// TIA Portal V20 export
FUNCTION_BLOCK "FB_Axis"   // FB30140, LAD
{ S7_Optimized_Access := 'TRUE' }
// stored: AutoNumber false, MemoryReserve 100, SetENOAutomatically false
   VAR_INPUT
      TO_PosAxis : TO_PositioningAxis;
      I_bMan_Enable : Bool;
      I_iHomeMode : Int;
      I_iHomePos : LReal;
   END_VAR
   VAR_IN_OUT
      Ds_Axis : "sAxis";
   END_VAR
   VAR
      instAxis01 { ExternalAccessible := 'False'; ExternalVisible := 'False'; ExternalWritable := 'False'} : "LAxisCtrl_PosAxis";
      instShearAxisStatus { S7_SetPoint := 'True'} : "LAxisCtrl_GetAxisStatusWord";
      RT_Reset { S7_SetPoint := 'True'} : R_TRIG;
      RT_PB { ExternalAccessible := 'False'; ExternalVisible := 'False'; ExternalWritable := 'False'} : Array[0..19] of R_TRIG;   // Störungen / Alarms
      FT_PB { ExternalAccessible := 'False'; ExternalVisible := 'False'; ExternalWritable := 'False'; S7_SetPoint := 'True'} : Array[0..19] of F_TRIG;   // Störungen unterdrücken, Belegung identisch mit "Alarm" / Hide Alarms, identical with "Alarm"
      TON_PB { ExternalAccessible := 'False'; ExternalVisible := 'False'; ExternalWritable := 'False'} : Array[0..19] of TON_TIME;   // Fallende Flanke / Falling edge
      TOF_PB { ExternalAccessible := 'False'; ExternalVisible := 'False'; ExternalWritable := 'False'} : Array[0..19] of TOF_TIME;   // Negativer Impuls / Negative pulse
      i { S7_SetPoint := 'True'} : Int;
      temp_cmd_bEnableAxis { ExternalAccessible := 'False'; ExternalVisible := 'False'; ExternalWritable := 'False'} : Bool;
      temp_cmd_bresetAxis { ExternalAccessible := 'False'; ExternalVisible := 'False'; ExternalWritable := 'False'} : Bool;
      temp_cmd_bjogForward { ExternalAccessible := 'False'; ExternalVisible := 'False'; ExternalWritable := 'False'} : Bool;
      temp_cmd_bjogBackward { ExternalAccessible := 'False'; ExternalVisible := 'False'; ExternalWritable := 'False'} : Bool;
      temp_cmd_bmoveVelocity { ExternalAccessible := 'False'; ExternalVisible := 'False'; ExternalWritable := 'False'} : Bool;
      temp_cmd_bstop { ExternalAccessible := 'False'; ExternalVisible := 'False'; ExternalWritable := 'False'} : Bool;
      temp_cmd_bfastStop { ExternalAccessible := 'False'; ExternalVisible := 'False'; ExternalWritable := 'False'} : Bool;
      temp_cmd_bhoming { ExternalAccessible := 'False'; ExternalVisible := 'False'; ExternalWritable := 'False'} : Bool;
      temp_cmd_bGoToPos { ExternalAccessible := 'False'; ExternalVisible := 'False'; ExternalWritable := 'False'} : Array[0..16] of Bool;
      temp_cmd_iGoToPos : Word;
      temp_cmd_bCallAbsPos : Bool;
      temp_cmd_bRelPos : Bool;
      temp_Para_rJog_Speed { ExternalAccessible := 'False'; ExternalVisible := 'False'; ExternalWritable := 'False'} : LReal;
      temp_cmd_bGoToPosAll { ExternalAccessible := 'False'; ExternalVisible := 'False'; ExternalWritable := 'False'} : Bool;
      temp_configuration { ExternalAccessible := 'False'; ExternalVisible := 'False'; ExternalWritable := 'False'} : "LAxisCtrl_typeAxisConfig";   // Diagnostics structure
      temp_Status { ExternalAccessible := 'False'; ExternalVisible := 'False'; ExternalWritable := 'False'} : Word;
      tempAxisEnabled { ExternalAccessible := 'False'; ExternalVisible := 'False'; ExternalWritable := 'False'} : Bool;
      temp_CommandBusy { ExternalAccessible := 'False'; ExternalVisible := 'False'; ExternalWritable := 'False'} : Bool;
      temp_CommandDone { ExternalAccessible := 'False'; ExternalVisible := 'False'; ExternalWritable := 'False'} : Bool;
      temp_CommandAborted { ExternalAccessible := 'False'; ExternalVisible := 'False'; ExternalWritable := 'False'} : Bool;
      temp_InVelocity { ExternalAccessible := 'False'; ExternalVisible := 'False'; ExternalWritable := 'False'} : Bool;
      temp_jogSelected { ExternalAccessible := 'False'; ExternalVisible := 'False'; ExternalWritable := 'False'} : Bool;
      tempPosAbsoluteSelected { ExternalAccessible := 'False'; ExternalVisible := 'False'; ExternalWritable := 'False'} : Bool;
      temp_diagnostics { ExternalAccessible := 'False'; ExternalVisible := 'False'; ExternalWritable := 'False'} : "LAxisCtrl_typeDiagnostics";
      temp_stop_Dec { ExternalAccessible := 'False'; ExternalVisible := 'False'; ExternalWritable := 'False'} : LReal;
      temp_faststop_Dec { ExternalAccessible := 'False'; ExternalVisible := 'False'; ExternalWritable := 'False'} : LReal;
      temp_iFBStatus : Word;
      temp_iMCStatus : Word;
      old_iFBStatus : Word;
      old_iMCStatus : Word;
   END_VAR
BEGIN

REGION Network 1
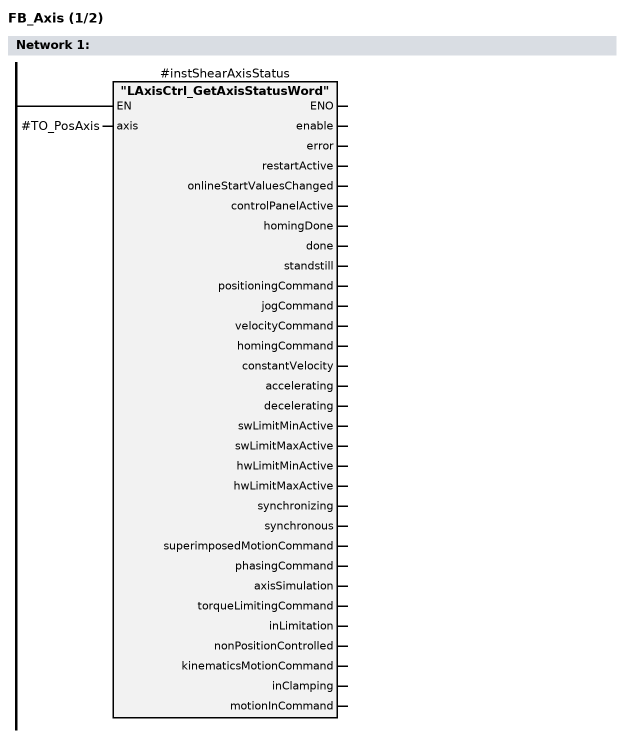
   RUNG wire#powerrail
      #instShearAxisStatus(axis := #TO_PosAxis, enable =>, error =>, restartActive =>, onlineStartValuesChanged =>, controlPanelActive =>, homingDone =>, done =>, standstill =>, positioningCommand =>, jogCommand =>, velocityCommand =>, homingCommand =>, constantVelocity =>, accelerating =>, decelerating =>, swLimitMinActive =>, swLimitMaxActive =>, hwLimitMinActive =>, hwLimitMaxActive =>, synchronizing =>, synchronous =>, superimposedMotionCommand =>, phasingCommand =>, axisSimulation =>, torqueLimitingCommand =>, inLimitation =>, nonPositionControlled =>, kinematicsMotionCommand =>, inClamping =>, motionInCommand =>)
   END_RUNG
   // the same network as SCL:
   #instShearAxisStatus(axis := #TO_PosAxis);   // "LAxisCtrl_GetAxisStatusWord"
END_REGION

REGION Network 2: LAxisCtrl
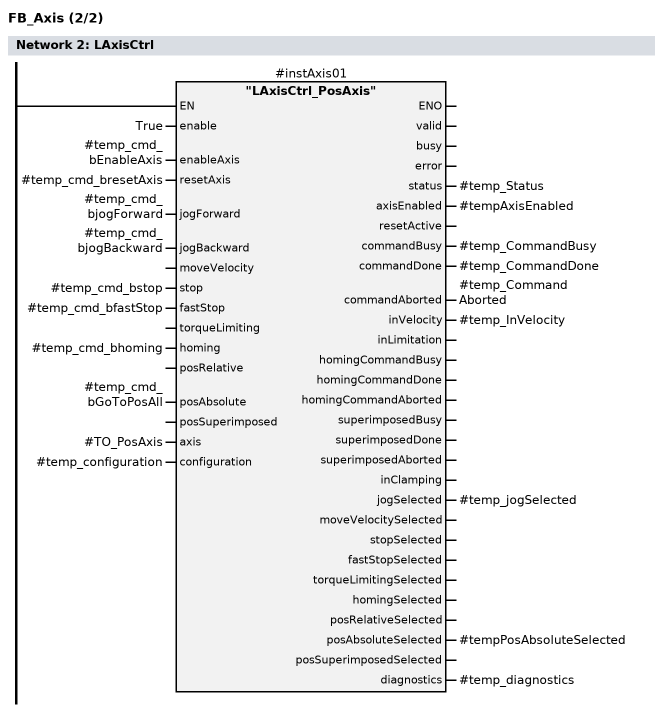
   RUNG wire#powerrail
      #instAxis01(enable := True, enableAxis := #temp_cmd_bEnableAxis, resetAxis := #temp_cmd_bresetAxis, jogForward := #temp_cmd_bjogForward, jogBackward := #temp_cmd_bjogBackward, moveVelocity :=, stop := #temp_cmd_bstop, fastStop := #temp_cmd_bfastStop, torqueLimiting :=, homing := #temp_cmd_bhoming, posRelative :=, posAbsolute := #temp_cmd_bGoToPosAll, posSuperimposed :=, axis := #TO_PosAxis, configuration := #temp_configuration, valid =>, busy =>, error =>, status => #temp_Status, axisEnabled => #tempAxisEnabled, resetActive =>, commandBusy => #temp_CommandBusy, commandDone => #temp_CommandDone, commandAborted => #temp_CommandAborted, inVelocity => #temp_InVelocity, inLimitation =>, homingCommandBusy =>, homingCommandDone =>, homingCommandAborted =>, superimposedBusy =>, superimposedDone =>, superimposedAborted =>, inClamping =>, jogSelected => #temp_jogSelected, moveVelocitySelected =>, stopSelected =>, fastStopSelected =>, torqueLimitingSelected =>, homingSelected =>, posRelativeSelected =>, posAbsoluteSelected => #tempPosAbsoluteSelected, posSuperimposedSelected =>, diagnostics => #temp_diagnostics)
   END_RUNG
   // the same network as SCL:
   #instAxis01(enable := True,   // "LAxisCtrl_PosAxis"
               enableAxis := #temp_cmd_bEnableAxis,
               resetAxis := #temp_cmd_bresetAxis,
               jogForward := #temp_cmd_bjogForward,
               jogBackward := #temp_cmd_bjogBackward,
               stop := #temp_cmd_bstop,
               fastStop := #temp_cmd_bfastStop,
               homing := #temp_cmd_bhoming,
               posAbsolute := #temp_cmd_bGoToPosAll,
               axis := #TO_PosAxis,
               configuration := #temp_configuration,
               status => #temp_Status,
               axisEnabled => #tempAxisEnabled,
               commandBusy => #temp_CommandBusy,
               commandDone => #temp_CommandDone,
               commandAborted => #temp_CommandAborted,
               inVelocity => #temp_InVelocity,
               jogSelected => #temp_jogSelected,
               posAbsoluteSelected => #tempPosAbsoluteSelected,
               diagnostics => #temp_diagnostics);
END_REGION

REGION Network 3 (SCL): input
   #temp_cmd_bEnableAxis  := #Ds_Axis.I_CMD.bEnableAxis OR (#Ds_Axis.I_HMI.bEnableAxis AND #I_bMan_Enable);
   #temp_cmd_bresetAxis   := #Ds_Axis.I_CMD.bResetAxis;
   #temp_cmd_bjogForward  := #Ds_Axis.I_InLock.bjogForward AND (#Ds_Axis.I_CMD.bjogForward OR (#Ds_Axis.I_HMI.bjogForward AND #I_bMan_Enable)) ;
   #temp_cmd_bjogBackward := #Ds_Axis.I_InLock.bjogBackward AND (#Ds_Axis.I_CMD.bjogBackward OR (#Ds_Axis.I_HMI.bjogBackward AND #I_bMan_Enable)) ;
   #temp_cmd_bstop        := #Ds_Axis.I_CMD.bstop OR (#Ds_Axis.I_HMI.bstop AND #I_bMan_Enable);
   #temp_cmd_bfastStop    := #Ds_Axis.I_CMD.bfastStop;
   #temp_cmd_bhoming      := #Ds_Axis.I_InLock.bHoming AND (#Ds_Axis.I_CMD.bHoming OR #Ds_Axis.I_HMI.bHoming) ;
END_REGION

REGION Network 4 (SCL): Configuration
   #Ds_Axis.I_Para.rJog_Speed[0] := 10.0;
   #Ds_Axis.I_Para.rMV_Speed[0] := 100.0;
   #Ds_Axis.I_Para.rStop_Dec[0] := 20.0;
   #Ds_Axis.I_Para.rEStop_Dec[0] := 50.0;

   #Ds_Axis.I_Para.rJog_Speed[1] := 100.0 * #Ds_Axis.I_Para.rJog_Speed[0];
   #Ds_Axis.I_Para.rJog_Speed[2] := 100.0 * #Ds_Axis.I_Para.rJog_Speed[0];
   #Ds_Axis.I_Para.rMV_Speed[1] := 100.0 * #Ds_Axis.I_Para.rMV_Speed[0];
   #Ds_Axis.I_Para.rMV_Speed[2] := 100.0 * #Ds_Axis.I_Para.rMV_Speed[0];
   #Ds_Axis.I_Para.rStop_Dec[1] := 100.0 * #Ds_Axis.I_Para.rStop_Dec[0];
   #Ds_Axis.I_Para.rEStop_Dec[1] := 100.0 * #Ds_Axis.I_Para.rEStop_Dec[0];

   IF #temp_configuration.jog.velocity <> #Ds_Axis.I_Para.rJog_Speed[0] OR
       #temp_configuration.jog.acceleration <> #Ds_Axis.I_Para.rJog_Speed[1] OR
       #temp_configuration.jog.deceleration <> #Ds_Axis.I_Para.rJog_Speed[2] OR
       #temp_configuration.moveVelocity.acceleration <> #Ds_Axis.I_Para.rMV_Speed[0] OR
       #temp_configuration.moveVelocity.deceleration <> #Ds_Axis.I_Para.rMV_Speed[1] OR
       #temp_configuration.moveVelocity.acceleration <> #Ds_Axis.I_Para.rMV_Speed[2] OR
       #temp_configuration.stop.deceleration <> #Ds_Axis.I_Para.rStop_Dec[0] OR
       #temp_configuration.stop.jerk <> #Ds_Axis.I_Para.rStop_Dec[1] OR
       #temp_configuration.fastStop.deceleration <> #Ds_Axis.I_Para.rEStop_Dec[0] OR
       #temp_configuration.fastStop.jerk <> #Ds_Axis.I_Para.rEStop_Dec[1]
   THEN
       // Jog
       #temp_configuration.jog.velocity := #Ds_Axis.I_Para.rJog_Speed[0];
       #temp_configuration.jog.acceleration := #Ds_Axis.I_Para.rJog_Speed[1];
       #temp_configuration.jog.deceleration := #Ds_Axis.I_Para.rJog_Speed[2];
       // Move
       #temp_configuration.moveVelocity.velocity := #Ds_Axis.I_Para.rMV_Speed[0];
       #temp_configuration.moveVelocity.acceleration := #Ds_Axis.I_Para.rMV_Speed[1];
       #temp_configuration.moveVelocity.deceleration := #Ds_Axis.I_Para.rMV_Speed[2];
       // Stop   
       #temp_configuration.stop.deceleration := #Ds_Axis.I_Para.rStop_Dec[0];
       #temp_configuration.stop.jerk := #Ds_Axis.I_Para.rStop_Dec[1];
       //faststoo
       #temp_configuration.fastStop.deceleration := #Ds_Axis.I_Para.rEStop_Dec[0];
       #temp_configuration.fastStop.jerk := #Ds_Axis.I_Para.rEStop_Dec[1];
   END_IF;

   // Homing
   #temp_configuration.homing.mode := #I_iHomeMode;//I_iHomeMode
   #temp_configuration.homing.position := #I_iHomePos;//I_iHomePos

   //AbsPos
   //#temp_cmd_bGoToPosAll := #Ds_Axis.I_CMD.bCallAbsPos AND #Ds_Axis.I_InLock.bGoToPos[1];//"dStruct_Axis".gs_Axis[0].I_CMD.bCallAbsPos
   #temp_cmd_bGoToPosAll := "dStruct_Axis".gs_Axis[0].I_HMI.bCallAbsPos AND #Ds_Axis.I_InLock.bGoToPos[1];
   //#temp_posAbsolute :=
   //#Ds_Axis.I_bGoToPos[0] OR #Ds_Axis.I_bGoToPos[1] OR #Ds_Axis.I_bGoToPos[2] OR #Ds_Axis.I_bGoToPos[3] OR
   //#Ds_Axis.I_bGoToPos[4] OR #Ds_Axis.I_bGoToPos[5] OR #Ds_Axis.I_bGoToPos[6] OR #Ds_Axis.I_bGoToPos[7] OR
   //#Ds_Axis.I_bGoToPos[8] OR #Ds_Axis.I_bGoToPos[9] OR #Ds_Axis.I_bGoToPos[10] OR #Ds_Axis.I_bGoToPos[11] OR
   //#Ds_Axis.I_bGoToPos[12] OR #Ds_Axis.I_bGoToPos[13] OR #Ds_Axis.I_bGoToPos[14] OR #Ds_Axis.I_bGoToPos[15];

   #temp_configuration.posAbsolute.position := "dStruct_Axis".gs_Axis[0].I_Para.rPos_Abs[0];//#Ds_Axis.I_Para.rPos_Abs[0];
   #temp_configuration.posAbsolute.velocity := "dStruct_Axis".gs_Axis[0].I_Para.rSpeed_Abs[0];//#Ds_Axis.I_Para.rSpeed_Abs[0];
   #temp_configuration.posAbsolute.direction := 3;

   #temp_configuration.posAbsolute.acceleration := #temp_configuration.posAbsolute.velocity * 10.0;//#Ds_Axis.Para.I_iAcc_Set;
   #temp_configuration.posAbsolute.deceleration := #temp_configuration.posAbsolute.velocity * 10.0;//#Ds_Axis.Para.I_iDec_Set;
   #temp_configuration.posAbsolute.jerk := #temp_configuration.posAbsolute.velocity * 100.0;//#Ds_Axis.Para.I_iJerk_Set;

   (*
   FOR #i := 0 TO 15 DO
   //    #RT_PB[#i](CLK := #Ds_Axis.I_bGoToPos[#i]);
       #RT_PB[#i](CLK := #Ds_Axis.CMD.I_bCallAbsPos);

       IF #RT_PB[#i].Q THEN
           #temp_configuration.posAbsolute.position := #Ds_Axis.Para.I_rPos_Abs[0];
           #temp_configuration.posAbsolute.velocity := #Ds_Axis.Para.I_rSpeed_Abs[0];
           #temp_configuration.posAbsolute.direction := 3;//temp_posAbsolute_direction

           #temp_configuration.posAbsolute.acceleration := #Ds_Axis.Para.I_iAcc_Set;
           #temp_configuration.posAbsolute.deceleration := #Ds_Axis.Para.I_iDec_Set;
           #temp_configuration.posAbsolute.jerk := #Ds_Axis.Para.I_iJerk_Set;

       END_IF;
   END_FOR;
   *)
END_REGION

REGION Network 5 (SCL): output
   #Ds_Axis.O_Status.bAxisEnabled := #tempAxisEnabled;
   #Ds_Axis.O_Status.bjogForward := #temp_cmd_bjogForward;//AND #temp_jogSelected ;
   #Ds_Axis.O_Status.bjogBackward := #temp_cmd_bjogBackward;//AND #temp_jogSelected;
   #Ds_Axis.O_Status.bHomed := #TO_PosAxis.StatusWord.%X5;
   #Ds_Axis.O_Status.bAxisError := #TO_PosAxis.StatusWord.%X1;
   #Ds_Axis.O_Status.rActPos := #TO_PosAxis.ActualPosition;
   #Ds_Axis.O_Status.rActSpeed := #TO_PosAxis.ActualVelocity;
   #Ds_Axis.O_Status.iAxisFaultNum := #TO_PosAxis.ErrorDetail.Number;
   //#Ds_Axis.O_DriveFaultNum
   //#Ds_Axis.O_Status.iFBStatus := #temp_diagnostics.status;
   //#Ds_Axis.O_Status.iMCStatus := #temp_diagnostics.subfunctionStatus;
   //#Ds_Axis.O_Torque
   //#Ds_Axis.oAxisName  := 


   #Ds_Axis.O_Status.bAtPos[0] := "FC_bNearIn"(rAct := #Ds_Axis.O_Status.rActPos, rTgt := #Ds_Axis.I_Para.rPos_Abs[0], rDelta := 1.0, bModule := 0, rModulo := 0);


   //#Ds_Axis.O_bPosDone
   //#Ds_Axis.O_bPosing
   //#tempPosAbsoluteSelected
END_REGION

REGION Network 6 (SCL): Reset
   #RT_Reset(CLK := #temp_cmd_bresetAxis);
   IF #RT_Reset.Q THEN
       #Ds_Axis.O_Status.iFBStatus := 16#00;
       #Ds_Axis.O_Status.iMCStatus := 16#00;
   END_IF;

   #temp_iFBStatus := #temp_diagnostics.status;
   IF #temp_iFBStatus <> #old_iFBStatus THEN
       #Ds_Axis.O_Status.iFBStatus := #temp_diagnostics.status;
       #old_iFBStatus := #temp_iFBStatus;
   END_IF;
   #temp_iMCStatus := #temp_diagnostics.subfunctionStatus;
   IF #temp_iMCStatus <> #old_iMCStatus THEN
       #Ds_Axis.O_Status.iFBStatus := #temp_diagnostics.subfunctionStatus;
       #old_iMCStatus := #temp_iMCStatus;
   END_IF;
END_REGION
END_FUNCTION_BLOCK
